// TIA Portal V17 export
// export: Created 2024-10-17T14:16:16.3399859Z, ExportSetting WithDefaults, DisplayName Totally Integrated Automation Portal, DisplayVersion V17 Update 4, DisplayName TIA Portal Openness, DisplayVersion V17 Update 4, DisplayName TIA Portal Version Control Interface, DisplayVersion V17, DisplayName SINAMICS Startdrive Advanced, DisplayVersion V17 Update2, DisplayName SINAMICS Startdrive G130, G150, S120, S150, SINAMICS MV, S210, DisplayVersion V17 Update2, DisplayName SINAMICS Startdrive G110M, G120, G120C, G120D, G120P, G115D, DisplayVersion V17 Update2, DisplayName STEP 7 Professional, DisplayVersion V17 Update 4, DisplayName STEP 7 Safety, DisplayVersion V17, DisplayName WinCC Advanced / Unified PC, DisplayVersion V17 Update 4
VAR_GLOBAL   // PLC tag table "LPMLV2022_PackTags_Constants"
END_VAR
VAR_GLOBAL CONSTANT   // user constants
   LPMLV2022_COMMAND_PARAMETER_BOOL_UPPER_LIM : UInt := 0;   // Size [0..UPPER_LIM] of structured Array of Unit/Machine Parameter information for values with BOOL data type
   LPMLV2022_COMMAND_PARAMETER_DINT_UPPER_LIM : UInt := 0;   // Size [0..UPPER_LIM] of structured Array of Unit/Machine Parameter information for values with DINT data type
   LPMLV2022_COMMAND_PARAMETER_REAL_UPPER_LIM : UInt := 0;   // Size [0..UPPER_LIM] of structured Array of Unit/Machine Parameter information for values with REAL data type
   LPMLV2022_COMMAND_PARAMETER_LREAL_UPPER_LIM : UInt := 0;   // Size [0..UPPER_LIM] of structured Array of Unit/Machine Parameter information for values with LREAL data type
   LPMLV2022_COMMAND_PARAMETER_STRING_UPPER_LIM : UInt := 0;   // Size [0..UPPER_LIM] of structured Array of Unit/Machine Parameter information for values with STRING data type
   LPMLV2022_COMMAND_RECIPE_UPPER_LIM : UInt := 0;   // Size [0..UPPER_LIM] of structured Array of Recipe Information
   LPMLV2022_COMMAND_PROCESS_VARIABLES_PARAMETER_BOOL_UPPER_LIM : UInt := 0;   // Size [0..UPPER_LIM] of structured Array of Recipe Process Variable information for values with BOOL data type
   LPMLV2022_COMMAND_PROCESS_VARIABLES_PARAMETER_DINT_UPPER_LIM : UInt := 0;   // Size [0..UPPER_LIM] of structured Array of Recipe Process Variable Information for values with DINT data type
   LPMLV2022_COMMAND_PROCESS_VARIABLES_PARAMETER_REAL_UPPER_LIM : UInt := 0;   // Size [0..UPPER_LIM] of structured Array of Recipe Process Variable information for values with REAL data type
   LPMLV2022_COMMAND_PROCESS_VARIABLES_PARAMETER_LREAL_UPPER_LIM : UInt := 0;   // Size [0..UPPER_LIM] of structured Array of Recipe Process Variable information for values with LREAL data type
   LPMLV2022_COMMAND_PROCESS_VARIABLES_PARAMETER_STRING_UPPER_LIM : UInt := 0;   // Size [0..UPPER_LIM] of structured Array of Recipe Process Variable information for values with STRING data type
   LPMLV2022_COMMAND_INGREDIENTS_PARAMETER_BOOL_UPPER_LIM : UInt := 0;   // Size [0..UPPER_LIM] of structured Array of Ingredient information for values with BOOL data type
   LPMLV2022_COMMAND_INGREDIENTS_PARAMETER_DINT_UPPER_LIM : UInt := 0;   // Size [0..UPPER_LIM] of structured Array of Ingredient Information for values with DINT data type
   LPMLV2022_COMMAND_INGREDIENTS_PARAMETER_REAL_UPPER_LIM : UInt := 0;   // Size [0..UPPER_LIM] of structured Array of Ingredient information for values with REAL data type
   LPMLV2022_COMMAND_INGREDIENTS_PARAMETER_LREAL_UPPER_LIM : UInt := 0;   // Size [0..UPPER_LIM] of structured Array of Ingredient information for values with LREAL data type
   LPMLV2022_COMMAND_INGREDIENTS_PARAMETER_STRING_UPPER_LIM : UInt := 0;   // Size [0..UPPER_LIM] of structured Array of Ingredient information for values with STRING data type
   LPMLV2022_STATUS_PARAMETER_BOOL_UPPER_LIM : UInt := 0;   // Size [0..UPPER_LIM] of structured Array of Unit/Machine Parameter information for values with BOOL data type
   LPMLV2022_STATUS_PARAMETER_DINT_UPPER_LIM : UInt := 0;   // Size [0..UPPER_LIM] of structured Array of Unit/Machine Parameter information for values with DINT data type
   LPMLV2022_STATUS_PARAMETER_REAL_UPPER_LIM : UInt := 0;   // Size [0..UPPER_LIM] of structured Array of Unit/Machine Parameter information for values with REAL data type
   LPMLV2022_STATUS_PARAMETER_LREAL_UPPER_LIM : UInt := 0;   // Size [0..UPPER_LIM] of structured Array of Unit/Machine Parameter information for values with LREAL data type
   LPMLV2022_STATUS_PARAMETER_STRING_UPPER_LIM : UInt := 0;   // Size [0..UPPER_LIM] of structured Array of Unit/Machine Parameter information for values with STRING data type
   LPMLV2022_STATUS_RECIPE_UPPER_LIM : UInt := 0;   // Size [0..UPPER_LIM] of structured Array of Recipe Information
   LPMLV2022_STATUS_PROCESS_VARIABLES_PARAMETER_BOOL_UPPER_LIM : UInt := 0;   // Size [0..UPPER_LIM] of structured Array of Recipe Process Variable information for values with BOOL data type
   LPMLV2022_STATUS_PROCESS_VARIABLES_PARAMETER_DINT_UPPER_LIM : UInt := 0;   // Size [0..UPPER_LIM] of structured Array of Recipe Process Variable Information for values with DINT data type
   LPMLV2022_STATUS_PROCESS_VARIABLES_PARAMETER_REAL_UPPER_LIM : UInt := 0;   // Size [0..UPPER_LIM] of structured Array of Recipe Process Variable information for values with REAL data type
   LPMLV2022_STATUS_PROCESS_VARIABLES_PARAMETER_LREAL_UPPER_LIM : UInt := 0;   // Size [0..UPPER_LIM] of structured Array of Recipe Process Variable information for values with LREAL data type
   LPMLV2022_STATUS_PROCESS_VARIABLES_PARAMETER_STRING_UPPER_LIM : UInt := 0;   // Size [0..UPPER_LIM] of structured Array of Recipe Process Variable information for values with STRING data type
   LPMLV2022_STATUS_INGREDIENTS_PARAMETER_BOOL_UPPER_LIM : UInt := 0;   // Size [0..UPPER_LIM] of structured Array of Ingredient information for values with BOOL data type
   LPMLV2022_STATUS_INGREDIENTS_PARAMETER_DINT_UPPER_LIM : UInt := 0;   // Size [0..UPPER_LIM] of structured Array of Ingredient Information for values with DINT data type
   LPMLV2022_STATUS_INGREDIENTS_PARAMETER_REAL_UPPER_LIM : UInt := 0;   // Size [0..UPPER_LIM] of structured Array of Ingredient information for values with REAL data type
   LPMLV2022_STATUS_INGREDIENTS_PARAMETER_LREAL_UPPER_LIM : UInt := 0;   // Size [0..UPPER_LIM] of structured Array of Ingredient information for values with LREAL data type
   LPMLV2022_STATUS_INGREDIENTS_PARAMETER_STRING_UPPER_LIM : UInt := 0;   // Size [0..UPPER_LIM] of structured Array of Ingredient information for values with STRING data type
   LPMLV2022_STATUS_STACK_LIGHT_UPPER_LIM : UInt := 0;   // Size [0..UPPER_LIM] of Indicator for the current stacklight status
   LPMLV2022_ADMIN_PARAMETER_BOOL_UPPER_LIM : UInt := 0;   // Size [0..UPPER_LIM] of structured Array of Unit/Machine Parameter information for values with BOOL data type
   LPMLV2022_ADMIN_PARAMETER_DINT_UPPER_LIM : UInt := 0;   // Size [0..UPPER_LIM] of structured Array of Unit/Machine Parameter information for values with DINT data type
   LPMLV2022_ADMIN_PARAMETER_REAL_UPPER_LIM : UInt := 0;   // Size [0..UPPER_LIM] of structured Array of Unit/Machine Parameter information for values with REAL data type
   LPMLV2022_ADMIN_PARAMETER_LREAL_UPPER_LIM : UInt := 0;   // Size [0..UPPER_LIM] of structured Array of Unit/Machine Parameter information for values with LREAL data type
   LPMLV2022_ADMIN_PARAMETER_STRING_UPPER_LIM : UInt := 0;   // Size [0..UPPER_LIM] of structured Array of Unit/Machine Parameter information for values with STRING data type
   LPMLV2022_ADMIN_ALARM_UPPER_LIM : UInt := 0;   // Size [0..UPPER_LIM] of Array for Machine Alarms
   LPMLV2022_ADMIN_ALARM_HISTORY_UPPER_LIM : UInt := 0;   // Size [0..UPPER_LIM] of Array for Machine Fault Number and Messaging History
   LPMLV2022_ADMIN_WARNING_UPPER_LIM : UInt := 0;   // Size [0..UPPER_LIM] of Machine warnings for general events that do not cause the machine to stop
   LPMLV2022_ADMIN_CUMULATIVE_TIMES_UPPER_LIM : UInt := 0;   // Size [0..UPPER_LIM] of structured Array of Timer Values
   LPMLV2022_ADMIN_NUMBER_OF_MODES_UPPER_LIM : UInt := 8;   // Size [0..UPPER_LIM] of structured Array of Mode and State Time Values for each Cumulative Time Tracker
   LPMLV2022_ADMIN_NUMBER_OF_STATES_UPPER_LIM : UInt := 17;   // Size [0..UPPER_LIM] of state Time Values for each State in each Mode
   LPMLV2022_ADMIN_PRODUCT_DATA_UPPER_LIM : UInt := 0;   // Size [0..UPPER_LIM] of structured array of Product Stream Data
END_VAR
